{attribute 'qualified_only'}
{attribute 'to_string'}
TYPE E_StepperStates :
(
	Idle:=0,
	Resetting,
	Homing1,
	Homing2,
	Disabled,
	Enabled,
	Jogging,
	MovingAbs,
	Halting
)UINT := Idle
;
END_TYPE

(* stored: Version 1.1.0.1, ProductVersion 3.1.4024.12
   EnumerationTextList E_StepperStates: Id {ff9491a3-2a18-46b4-a15e-988191356dfb} *)
